TYPE ST_Identity_PK4_OUT2 :
STRUCT
	ID	:STRING;
	ReadQuality:STRING;
END_STRUCT
END_TYPE

(* stored: Version 1.1.0.1, ProductVersion 3.1.4024.13
   DUT ST_Identity_PK4_OUT2: Id {95bf2ce3-3de5-4761-82da-1bb504481650} *)
